// TIA Portal V20 export
DATA_BLOCK "Config"   // DB151
// stored: MemoryReserve 100, Namespace Unit1.Em11
   VAR
      em : "LAF_typeEmConfiguration";   // Configuration of EM Parameters
      cmWeightCheckJRDetect : "LBC_typeDigitalSignalConfiguration";
      cmWeightCheckControl : "LER_WeightCheckConfiguration";
      "=====미사용=====" { ExternalAccessible := 'False'; ExternalVisible := 'False'; ExternalWritable := 'False'} : Bool;
      cmWeightCheckStageLiftUpDown : "LBC_typeTwoWayActuatorConfiguration";
   END_VAR
BEGIN
   em.referenceDesignator.parent := WSTRING#'U1';
   em.referenceDesignator.relative := WSTRING#'EM0';
   cmWeightCheckControl.hwID.pncMainControlID := 612;
   cmWeightCheckControl.hwID.pncMainStatusID := 612;
   cmWeightCheckControl.hwID.scaleControlID := 613;
   cmWeightCheckControl.hwID.scaleStatusID := 613;
END_DATA_BLOCK
